// TIA Portal V20 export
TYPE "typeSequenceControlNode_sideTapeAttachment"
// stored: Namespace Unit1.Em4
   STRUCT
      jobs : "LAF_typeJobs";
      sequence : "LAF_typeSequence";
      selectJobStatus { S7_SetPoint := 'True'} : Array[0..10] of "LAF_typeJobStatus";
      "step" : "LER_typeStep";
      jobInterface : "Unit1.Em4.typeSequenceControlNodeJobInterface_sideTapeAttachment";
      homeCheck : "Unit1.Em4.typeSequenceControlNodeHomeCheck_sideTapeAttachment";
   END_STRUCT;
   // // "step".action1[101] : Step[101] : JOB[1] Condition
   // // "step".action1[110] : Step[110] : Side Tape Attachment Left, Right Backward
   // // "step".action1[111] : Step[111] : Side Tape Attachment Y-Axis Wait Pos
   // // "step".action1[120] : Step[120] : Side Tape Attachment Bottom Forward
   // // "step".action1[130] : Step[130] : Side Tape Attachment Remain Attach Left Condition
   // // "step".action1[131] : Step[131] : Side Tape Attachment X-Axis Remain Attach Left Position
   // // "step".action1[132] : Step[132] : Side Tape Attachment Y-Axis Remain Attach Left Position
   // // "step".action1[133] : Step[133] : Side Tape Attachment Left Vaccum Off
   // // "step".action1[134] : Step[134] : Side Tape Attachment Y-Axis Wait Pos
   // // "step".action1[140] : Step[140] : Side Tape Attachment Remain Attach Right Condition
   // // "step".action1[141] : Step[141] : Side Tape Attachment X-Axis Remain Attach Right Position
   // // "step".action1[142] : Step[142] : Side Tape Attachment Y-Axis Remain Attach Right Position
   // // "step".action1[143] : Step[143] : Side Tape Attachment Right Vaccum Off
   // // "step".action1[144] : Step[144] : Side Tape Attachment Y-Axis Wait Pos
   // // "step".action1[180] : Step[180] : Side Tape Attachment X-Axis Wait Position
   // // "step".action1[190] : Step[190] : Job[1] Step End
   // // "step".action1[201] : Step[201] : JOB[2] Condition
   // // "step".action1[210] : Step[210] : Side Tape Attachment X-Axis Right Loading Pos
   // // "step".action1[220] : Step[220] : Side Tape Attachment Y-Axis Loading Pos
   // // "step".action1[221] : Step[221] : Side Tape Attachment-2 Vaccum On
   // // "step".action1[230] : Step[230] : Side Tape Cutter Forward
   // // "step".action1[231] : Step[231] : Side Tape Cutter Backward
   // // "step".action1[240] : Step[240] : Side Tape Clamp Open
   // // "step".action1[241] : Step[241] : Spare
   // // "step".action1[270] : Step[270] : Side Tape Attachment Y-Axis Wait Pos
   // // "step".action1[280] : Step[280] : Side Tape Attachment X-Axis Wait Pos
   // // "step".action1[290] : Step[290] : Job[2] Step End
   // // "step".action1[301] : Step[301] : JOB[3] Condition
   // // "step".action1[310] : Step[310] : Side Tape Attachment X-Axis Left Loading Pos
   // // "step".action1[320] : Step[320] : Side Tape Attachment Y-Axis Loading Pos
   // // "step".action1[321] : Step[321] : Side Tape Attachment-1 Vaccum On
   // // "step".action1[330] : Step[330] : Side Tape Cutter Forward
   // // "step".action1[331] : Step[331] : Side Tape Cutter Backward
   // // "step".action1[340] : Step[340] : Side Tape Clamp Open
   // // "step".action1[341] : Step[341] : Spare
   // // "step".action1[370] : Step[370] : Side Tape Attachment Y-Axis Wait Pos
   // // "step".action1[380] : Step[380] : Side Tape Attachment X-Axis Tape-1 Put Pos
   // // "step".action1[390] : Step[390] : Job[3] Step End
   // // "step".action1[401] : Step[401] : JOB[4] Condition
   // // "step".action1[410] : Step[410] : Side Tape Attachment X-Axis Tape-1 Put Pos
   // // "step".action1[420] : Step[420] : Side tape Attachment Y-Axis Tape-1 Put Pos
   // // "step".action1[421] : Step[421] : Side Tape Attachment Left, Right Forward, Vaccum Off
   // // "step".action1[422] : Step[422] : Spare
   // // "step".action1[430] : Step[430] : Side Tape Attachment Left, Right Backward
   // // "step".action1[431] : Step[431] : Side Tape Attachment Y-Axis Wait Pos
   // // "step".action1[480] : Step[480] : Side Tape Attachment X-Axis Wait Pos
   // // "step".action1[490] : Step[490] : Job[4] Step End
   // // "step".action1[501] : Step[501] : Job[5] Condition
   // // "step".action1[510] : Step[510] : Side Tape Attachment X-Axis Tape-2 Put Pos
   // // "step".action1[520] : Step[520] : Side tape Attachment Y-Axis Tape-2 Put Pos
   // // "step".action1[521] : Step[521] : Side Tape Attachment Right Forward, Vaccum Off
   // // "step".action1[522] : Step[522] : Spare
   // // "step".action1[530] : Step[530] : Side Tape Attachment Right Backward
   // // "step".action1[531] : Step[531] : Side Tape Attachment Y-Axis Wait Pos
   // // "step".action1[580] : Step[580] : Side Tape Attachment X-Axis Wait Pos
   // // "step".action1[590] : Step[590] : Job[5] Step End
   // // "step".action1[601] : Step[601] : Job[6] Condition
   // // "step".action1[610] : Step[610] : Side Tape Attachment X-Axis Tape-3 Put Pos
   // // "step".action1[620] : Step[620] : Side tape Attachment Y-Axis Tape-2 Put Pos
   // // "step".action1[621] : Step[621] : Side Tape Attachment Right Forward, Vaccum Off
   // // "step".action1[622] : Step[622] : Spare
   // // "step".action1[630] : Step[630] : Side Tape Attachment Right Backward
   // // "step".action1[631] : Step[631] : Side Tape Attachment Y-Axis Wait Pos
   // // "step".action1[680] : Step[680] : Side Tape Attachment X-Axis Wait Pos
   // // "step".action1[690] : Step[690] : Job[6] Step End
   // // "step".action1[701] : Step[701] : Job[7] Condition
   // // "step".action1[710] : Step[710] : Side Tape Attachment X-Axis Tape-4 Put Pos
   // // "step".action1[720] : Step[720] : Side tape Attachment Y-Axis Tape-1 Put Pos
   // // "step".action1[721] : Step[721] : Side Tape Attachment Right Forward, Vaccum Off
   // // "step".action1[722] : Step[722] : Spare
   // // "step".action1[730] : Step[730] : Side Tape Attachment Right Backward
   // // "step".action1[731] : Step[731] : Side Tape Attachment Y-Axis Wait Pos
   // // "step".action1[780] : Step[780] : Side Tape Attachment X-Axis Wait Pos
   // // "step".action1[790] : Step[790] : Job[7] Step End
   // // "step".transition1[101] : Step[101] : JOB[1] Condition
   // // "step".transition1[110] : Step[110] : Side Tape Attachment Left, Right Backward
   // // "step".transition1[111] : Step[111] : Side Tape Attachment Y-Axis Wait Pos
   // // "step".transition1[180] : Step[180] : Side Tape Attachment Bottom Forward
   // // "step".transition1[181] : Step[181] : Side Tape Attachment X-Axis Wait Position
   // // "step".transition1[190] : Step[190] : Job[1] Step End
   // // "step".transition1[201] : Step[201] : JOB[2] Condition
   // // "step".transition1[210] : Step[210] : Side Tape Attachment X-Axis Right Loading Pos
   // // "step".transition1[220] : Step[220] : Side Tape Attachment Y-Axis Loading Pos
   // // "step".transition1[221] : Step[221] : Side Tape Attachment-2 Vaccum On
   // // "step".transition1[230] : Step[230] : Side Tape Cutter Forward
   // // "step".transition1[231] : Step[231] : Side Tape Cutter Backward
   // // "step".transition1[240] : Step[240] : Side Tape Clamp Open
   // // "step".transition1[241] : Step[241] : Spare
   // // "step".transition1[270] : Step[270] : Side Tape Attachment Y-Axis Wait Pos
   // // "step".transition1[280] : Step[280] : Side Tape Attachment X-Axis Wait Pos
   // // "step".transition1[290] : Step[290] : Job[2] Step End
   // // "step".transition1[301] : Step[301] : JOB[3] Condition
   // // "step".transition1[310] : Step[310] : Side Tape Attachment X-Axis Left Loading Pos
   // // "step".transition1[320] : Step[320] : Side Tape Attachment Y-Axis Loading Pos
   // // "step".transition1[321] : Step[321] : Side Tape Attachment-1 Vaccum On
   // // "step".transition1[330] : Step[330] : Side Tape Cutter Forward
   // // "step".transition1[331] : Step[331] : Side Tape Cutter Backward
   // // "step".transition1[340] : Step[340] : Side Tape Clamp Open
   // // "step".transition1[341] : Step[341] : Spare
   // // "step".transition1[370] : Step[370] : Side Tape Attachment Y-Axis Wait Pos
   // // "step".transition1[380] : Step[380] : Side Tape Attachment X-Axis Tape-1 Put Pos
   // // "step".transition1[390] : Step[390] : Job[3] Step End
   // // "step".transition1[401] : Step[401] : JOB[4] Condition
   // // "step".transition1[410] : Step[410] : Side Tape Attachment X-Axis Tape-1 Put Pos
   // // "step".transition1[420] : Step[420] : Side tape Attachment Y-Axis Tape-1 Put Pos
   // // "step".transition1[421] : Step[421] : Side Tape Attachment Left, Right Forward, Vaccum Off
   // // "step".transition1[422] : Step[422] : Spare
   // // "step".transition1[430] : Step[430] : Side Tape Attachment Left, Right Backward
   // // "step".transition1[431] : Step[431] : Side Tape Attachment Y-Axis Wait Pos
   // // "step".transition1[480] : Step[480] : Side Tape Attachment X-Axis Wait Pos
   // // "step".transition1[490] : Step[490] : Job[4] Step End
   // // "step".transition1[501] : Step[501] : Job[5] Condition
   // // "step".transition1[510] : Step[510] : Side Tape Attachment X-Axis Tape-2 Put Pos
   // // "step".transition1[520] : Step[520] : Side tape Attachment Y-Axis Tape-2 Put Pos
   // // "step".transition1[521] : Step[521] : Side Tape Attachment Right Forward, Vaccum Off
   // // "step".transition1[522] : Step[522] : Spare
   // // "step".transition1[530] : Step[530] : Side Tape Attachment Right Backward
   // // "step".transition1[531] : Step[531] : Side Tape Attachment Y-Axis Wait Pos
   // // "step".transition1[580] : Step[580] : Side Tape Attachment X-Axis Wait Pos
   // // "step".transition1[590] : Step[590] : Job[5] Step End
   // // "step".transition1[601] : Step[601] : Job[6] Condition
   // // "step".transition1[610] : Step[610] : Side Tape Attachment X-Axis Tape-3 Put Pos
   // // "step".transition1[620] : Step[620] : Side tape Attachment Y-Axis Tape-2 Put Pos
   // // "step".transition1[621] : Step[621] : Side Tape Attachment Right Forward, Vaccum Off
   // // "step".transition1[622] : Step[622] : Spare
   // // "step".transition1[630] : Step[630] : Side Tape Attachment Right Backward
   // // "step".transition1[631] : Step[631] : Side Tape Attachment Y-Axis Wait Pos
   // // "step".transition1[680] : Step[680] : Side Tape Attachment X-Axis Wait Pos
   // // "step".transition1[690] : Step[690] : Job[6] Step End
   // // "step".transition1[701] : Step[701] : Job[7] Condition
   // // "step".transition1[710] : Step[710] : Side Tape Attachment X-Axis Tape-4 Put Pos
   // // "step".transition1[720] : Step[720] : Side tape Attachment Y-Axis Tape-1 Put Pos
   // // "step".transition1[721] : Step[721] : Side Tape Attachment Right Forward, Vaccum Off
   // // "step".transition1[722] : Step[722] : Spare
   // // "step".transition1[730] : Step[730] : Side Tape Attachment Right Backward
   // // "step".transition1[731] : Step[731] : Side Tape Attachment Y-Axis Wait Pos
   // // "step".transition1[780] : Step[780] : Side Tape Attachment X-Axis Wait Pos
   // // "step".transition1[790] : Step[790] : Job[7] Step End
END_TYPE
